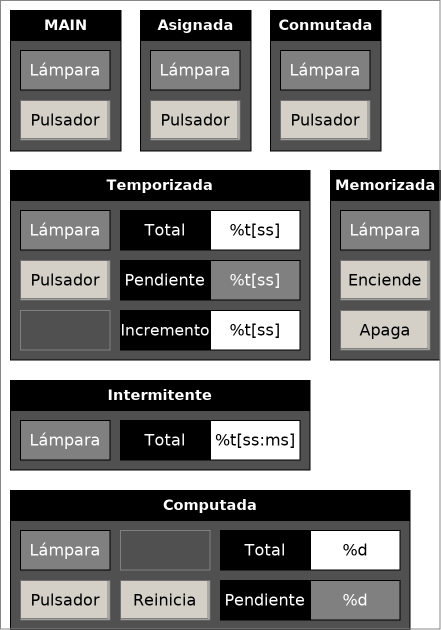
VISUALIZATION VISU_Lampara  // 441x630
    Rectangle (10,40 111x111)
    Rectangle (20,50 90x40), "Lámpara", colour toggle: MAIN.Lampara
    Button (20,100 90x40), "Pulsador"
        tap MAIN.Pulsador
    Rectangle (10,10 111x30), "MAIN"
    Rectangle (10,200 300x160)
    Rectangle (20,210 90x40), "Lámpara", colour toggle: MAIN.LamparaTemporizada.Lampara
    Button (20,260 90x40), "Pulsador"
        tap MAIN.LamparaTemporizada.Pulsador
    Rectangle (10,170 300x30), "Temporizada"
    Rectangle (120,210 90x40), "Total"
    Rectangle (210,210 90x40), "%t[ss]", text variable: MAIN.LamparaTemporizada.TiempoEncendido
        OnMouseDown: write the text variable via Default
    Rectangle (120,260 90x40), "Pendiente"
    Rectangle (210,260 90x40), "%t[ss]", text variable: MAIN.LamparaTemporizada.TiempoPendiente
    Rectangle (140,40 111x111)
    Rectangle (150,50 90x40), "Lámpara", colour toggle: MAIN.LamparaAsignada.Lampara
    Button (150,100 90x40), "Pulsador"
        tap MAIN.LamparaAsignada.Pulsador
    Rectangle (140,10 111x30), "Asignada"
    Rectangle (270,40 111x111)
    Rectangle (280,50 90x40), "Lámpara", colour toggle: MAIN.LamparaConmutada.Lampara
    Button (280,100 90x40), "Pulsador"
        tap MAIN.LamparaConmutada.Pulsador
    Rectangle (270,10 111x30), "Conmutada"
    Rectangle (10,520 400x110)
    Rectangle (20,530 90x40), "Lámpara", colour toggle: MAIN.LamparaComputada.Lampara
    Button (20,580 90x40), "Pulsador"
        tap MAIN.LamparaComputada.Pulsador
    Rectangle (10,490 400x30), "Computada"
    Rectangle (220,530 90x40), "Total"
    Rectangle (310,530 90x40), "%d", text variable: MAIN.LamparaComputada.ManiobrasTotales
        OnMouseDown: write the text variable via Default
    Rectangle (220,580 90x40), "Pendiente"
    Rectangle (310,580 90x40), "%d", text variable: MAIN.LamparaComputada.ManiobrasPendientes
    Button (120,580 90x40), "Reinicia"
        tap MAIN.LamparaComputada.PulsadorReinicio
    Rectangle (330,200 110x160)
    Rectangle (340,210 90x40), "Lámpara", colour toggle: MAIN.LamparaMemorizada.Lampara
    Button (340,310 90x40), "Apaga"
        tap MAIN.LamparaMemorizada.PulsadorDesconexion
    Rectangle (330,170 111x30), "Memorizada"
    Button (340,260 90x40), "Enciende"
        tap MAIN.LamparaMemorizada.PulsadorConexion
    Rectangle (10,410 300x60)
    Rectangle (20,420 90x40), "Lámpara", colour toggle: MAIN.LamparaIntermitente.Lampara
    Rectangle (10,380 300x30), "Intermitente"
    Rectangle (120,420 90x40), "Total"
    Rectangle (210,420 90x40), "%t[ss:ms]", text variable: MAIN.LamparaIntermitente.TiempoParpadeo
        OnMouseDown: write the text variable via Default
    Rectangle (120,310 90x40), "Incremento"
    Rectangle (210,310 90x40), "%t[ss]", text variable: MAIN.LamparaTemporizada.IncrementoTiempo
        OnMouseDown: write the text variable via Default
    Rectangle (120,530 90x40)
    Rectangle (20,310 90x40)
END_VISUALIZATION

(* stored: Version 1.1.0.1, ProductVersion 3.1.4024.15
   Visu VISU_Lampara: Id {9c96670d-5611-45f7-b475-36643b25dd97} *)
